{attribute 'GeneratedUsingTerminal: EL9010--0000'}
{attribute addProperty BoxType "EL9010--0000"}
{attribute addProperty Description "EL9010 End Terminal"}
{attribute addProperty Physics "K"}
{attribute addProperty Id "EL9010"}
{attribute addProperty CRC "3533447301"}
{attribute addProperty Size "0"}
TYPE EL9010_D29C2085 EXTENDS EtcSlaveTerminalBase_947E5A46 :
STRUCT
END_STRUCT
END_TYPE

(* stored: Version 1.2.0.0, ProductVersion 3.1.4024.9
   DUT EL9010_D29C2085: Id {ea3cc929-277a-430e-b34e-9efa2080993c} *)
